FUNCTION_BLOCK A21Alarms
VAR_OUTPUT
	panelPowerOn : BOOL;
	safetyOk : BOOL;
	airPressureOk : BOOL;
END_VAR
VAR_OUTPUT
	alarm : BOOL;
END_VAR

alarm :=
	NOT panelPowerOn OR 
	NOT safetyOk OR
	NOT airPressureOk;

END_FUNCTION_BLOCK

(* stored: Version 1.1.0.1, ProductVersion 3.1.4024.11
   POU A21Alarms: Id {52cc73a4-5d87-414b-9f82-1691c8b1fc45}, SpecialFunc None *)
